RoomTemp_198();
TempAdjust_198();
FilterSign_198();
FilterSignReset_198();
RemoteControlStart_198();

RemoteControlTempAdjust_198();












StartStopCommand_199();
StartStopStatus_199();
Alarm_199();
MalfunctionCode_199();




RoomTemp_199();
TempAdjust_199();
FilterSign_199();
FilterSignReset_199();
RemoteControlStart_199();

RemoteControlTempAdjust_199();












StartStopCommand_200();
StartStopStatus_200();
Alarm_200();
MalfunctionCode_200();




RoomTemp_200();
TempAdjust_200();
FilterSign_200();
FilterSignReset_200();
RemoteControlStart_200();

RemoteControlTempAdjust_200();












StartStopCommand_201();
StartStopStatus_201();
Alarm_201();
MalfunctionCode_201();




RoomTemp_201();
TempAdjust_201();
FilterSign_201();
FilterSignReset_201();
RemoteControlStart_201();

RemoteControlTempAdjust_201();












StartStopCommand_202();
StartStopStatus_202();
Alarm_202();
MalfunctionCode_202();




RoomTemp_202();
TempAdjust_202();
FilterSign_202();
FilterSignReset_202();
RemoteControlStart_202();

RemoteControlTempAdjust_202();












StartStopCommand_203();
StartStopStatus_203();
Alarm_203();
MalfunctionCode_203();




RoomTemp_203();
TempAdjust_203();
FilterSign_203();
FilterSignReset_203();
RemoteControlStart_203();

RemoteControlTempAdjust_203();












StartStopCommand_204();
StartStopStatus_204();
Alarm_204();
MalfunctionCode_204();




RoomTemp_204();
TempAdjust_204();
FilterSign_204();
FilterSignReset_204();
RemoteControlStart_204();

RemoteControlTempAdjust_204();












StartStopCommand_205();
StartStopStatus_205();
Alarm_205();
MalfunctionCode_205();




RoomTemp_205();
TempAdjust_205();
FilterSign_205();
FilterSignReset_205();
RemoteControlStart_205();

RemoteControlTempAdjust_205();












StartStopCommand_206();
StartStopStatus_206();
Alarm_206();
MalfunctionCode_206();




RoomTemp_206();
TempAdjust_206();
FilterSign_206();
FilterSignReset_206();
RemoteControlStart_206();

RemoteControlTempAdjust_206();












StartStopCommand_207();
StartStopStatus_207();
Alarm_207();
MalfunctionCode_207();




RoomTemp_207();
TempAdjust_207();
FilterSign_207();
FilterSignReset_207();
RemoteControlStart_207();

RemoteControlTempAdjust_207();












StartStopCommand_208();
StartStopStatus_208();
Alarm_208();
MalfunctionCode_208();




RoomTemp_208();
TempAdjust_208();
FilterSign_208();
FilterSignReset_208();
RemoteControlStart_208();

RemoteControlTempAdjust_208();












StartStopCommand_209();
StartStopStatus_209();
Alarm_209();
MalfunctionCode_209();




RoomTemp_209();
TempAdjust_209();
FilterSign_209();
FilterSignReset_209();
RemoteControlStart_209();

RemoteControlTempAdjust_209();












StartStopCommand_210();
StartStopStatus_210();
Alarm_210();
MalfunctionCode_210();




RoomTemp_210();
TempAdjust_210();
FilterSign_210();
FilterSignReset_210();
RemoteControlStart_210();

RemoteControlTempAdjust_210();












StartStopCommand_211();
StartStopStatus_211();
Alarm_211();
MalfunctionCode_211();




RoomTemp_211();
TempAdjust_211();
FilterSign_211();
FilterSignReset_211();
RemoteControlStart_211();

RemoteControlTempAdjust_211();












StartStopCommand_212();
StartStopStatus_212();
Alarm_212();
MalfunctionCode_212();




RoomTemp_212();
TempAdjust_212();
FilterSign_212();
FilterSignReset_212();
RemoteControlStart_212();

RemoteControlTempAdjust_212();












StartStopCommand_213();
StartStopStatus_213();
Alarm_213();
MalfunctionCode_213();




RoomTemp_213();
TempAdjust_213();
FilterSign_213();
FilterSignReset_213();
RemoteControlStart_213();

RemoteControlTempAdjust_213();












StartStopCommand_224();
StartStopStatus_224();
Alarm_224();
MalfunctionCode_224();




RoomTemp_224();
TempAdjust_224();
FilterSign_224();
FilterSignReset_224();
RemoteControlStart_224();

RemoteControlTempAdjust_224();












StartStopCommand_225();
StartStopStatus_225();
Alarm_225();
MalfunctionCode_225();




RoomTemp_225();
TempAdjust_225();
FilterSign_225();
FilterSignReset_225();
RemoteControlStart_225();

RemoteControlTempAdjust_225();












StartStopCommand_226();
StartStopStatus_226();
Alarm_226();
MalfunctionCode_226();




RoomTemp_226();
TempAdjust_226();
FilterSign_226();
FilterSignReset_226();
RemoteControlStart_226();

RemoteControlTempAdjust_226();












StartStopCommand_227();
StartStopStatus_227();
Alarm_227();
MalfunctionCode_227();




RoomTemp_227();
TempAdjust_227();
FilterSign_227();
FilterSignReset_227();
RemoteControlStart_227();

RemoteControlTempAdjust_227();












StartStopCommand_241();
StartStopStatus_241();
Alarm_241();
MalfunctionCode_241();




RoomTemp_241();
TempAdjust_241();
FilterSign_241();
FilterSignReset_241();
RemoteControlStart_241();

RemoteControlTempAdjust_241();












CL_Rejection_000();
SystemForcedOff_000();
CL_Rejection_064();
SystemForcedOff_064();
CL_Rejection_128();
SystemForcedOff_128();
CL_Rejection_192();
SystemForcedOff_192();

END_FUNCTION_BLOCK

(* stored: Version 1.1.0.1, ProductVersion 3.1.4024.14
   POU FB_BACnet_DAIKIN_MasterStation_III_No_9: Id {78cb49fc-2518-4e04-8b17-bd02b4a8e0e4}, SpecialFunc None *)
